Fanuc KAREL source: kt00748.KL

-- PROVISIONAL review KL for V1013-1; original PC SHA256 945f1c6ed56853f29e8a976c560ffdc8c549b69165bc032566c36e0666c23091
-- Incomplete behavior may be omitted. Consult companion uncertainty JSON. Do not deploy.
PROGRAM KT00748
%NOLOCKGROUP
VAR
  I1 : INTEGER
  I2 : INTEGER
  OUT : INTEGER
BEGIN
  -- UNRESOLVED_PC offsets 5-16; opcodes 2E,23
  -- UNRESOLVED_PC offsets 21-32; opcodes 2E,23
  -- UNRESOLVED_PC offsets 37-48; opcodes 2E,23
  -- UNRESOLVED_PC offsets 53-64; opcodes 2E,23
  -- UNRESOLVED_PC offsets 69-82; opcodes 21,50,23
  -- UNRESOLVED_PC offsets 87-91; opcodes 7F
END KT00748
